// TIA Portal V20 export
VAR_GLOBAL   // PLC tag table "Cabinet_15"
   iSz15_Actuator_Down AT %I5000.0 : Bool;
   iSz15_Actuator_Up AT %I5000.1 : Bool;
   oSz15_Pneumatic_Unit AT %Q5000.0 : Bool;
   oSz15_Actuator_Push AT %Q5000.1 : Bool;
   oSz15_Actuator_Pull AT %Q5000.2 : Bool;
   iSz15_Key_ON AT %I5000.2 : Bool;
   iSz15_Key_OFF AT %I5000.3 : Bool;
END_VAR
